INTERFACE I_ToString EXTENDS I_Base

METHOD ToString : T_MaxString
VAR_INPUT
END_VAR
END_METHOD

END_INTERFACE

(* stored: Version 1.1.0.1, ProductVersion 3.1.4026.18
   Itf I_ToString: Id {242b2e03-8ac7-0032-3400-3ad8a437b02d}
   Method ToString: Id {3c71be8f-ab57-0678-20c3-96c819817922} *)
